FUNCTION_BLOCK StopAllComponentsVisitor IMPLEMENTS I_ComponentVisitor
VAR
	Stoppable : I_Stoppable;
	_Stopped  : BOOL;
END_VAR

METHOD Stop
VAR_INPUT
	Components : I_ComponentCollection;
END_VAR
_Stopped := TRUE;
Components.Accept(THIS^);
END_METHOD

{attribute 'monitoring' := 'call'}
PROPERTY Stopped : BOOL
GET
Stopped := _Stopped;
END_GET
END_PROPERTY

METHOD VisitComponent
VAR_INPUT
	Component : I_Component;
END_VAR
IF __QUERYINTERFACE(Component, Stoppable) THEN
	Stoppable.Stop();
	IF NOT Stoppable.Stopped THEN
		_Stopped := FALSE;
	END_IF
END_IF
END_METHOD

END_FUNCTION_BLOCK

(* stored: Version 1.1.0.1, ProductVersion 3.1.4026.18
   POU StopAllComponentsVisitor: Id {ee4ec0b3-4c2a-44b2-a6fe-73a91a90a035}, SpecialFunc None
   Method Stop: Id {1bfd48af-b250-4fc3-a57c-055b0603f97a}
   Property Stopped: Id {2a33b24c-acd4-4d13-aa3e-46988a89de90}
   Get Get: Id {f65a0f1d-6f58-41a8-a1d0-71f0f99f2532}
   Method VisitComponent: Id {267eea54-520f-4c73-9c11-e182033c07b1} *)
